{attribute addProperty BoxType "KL2809"}
{attribute addProperty Id "Channel_1Channel_E75BD82E00Channel_2Channel_E75BD82E00Channel_3Channel_E75BD82E00Channel_4Channel_E75BD82E00Channel_5Channel_E75BD82E00Channel_6Channel_E75BD82E00Channel_7Channel_E75BD82E00Channel_8Channel_E75BD82E00Channel_9Channel_E75BD82E00Channel_10Channel_E75BD82E00Channel_11Channel_E75BD82E00Channel_12Channel_E75BD82E00Channel_13Channel_E75BD82E00Channel_14Channel_E75BD82E00Channel_15Channel_E75BD82E00Channel_16Channel_E75BD82E00"}
{attribute addProperty CRC "944202743"}
{attribute addProperty SizeInBites "0"}
{attribute addProperty SizeInBytes "0"}
TYPE KL2809_384763F7 :
STRUCT
	{attribute addProperty Name "Channel_1"}
	Channel_1 : Channel_E75BD82E;
	{attribute addProperty Name "Channel_2"}
	Channel_2 : Channel_E75BD82E;
	{attribute addProperty Name "Channel_3"}
	Channel_3 : Channel_E75BD82E;
	{attribute addProperty Name "Channel_4"}
	Channel_4 : Channel_E75BD82E;
	{attribute addProperty Name "Channel_5"}
	Channel_5 : Channel_E75BD82E;
	{attribute addProperty Name "Channel_6"}
	Channel_6 : Channel_E75BD82E;
	{attribute addProperty Name "Channel_7"}
	Channel_7 : Channel_E75BD82E;
	{attribute addProperty Name "Channel_8"}
	Channel_8 : Channel_E75BD82E;
	{attribute addProperty Name "Channel_9"}
	Channel_9 : Channel_E75BD82E;
	{attribute addProperty Name "Channel_10"}
	Channel_10 : Channel_E75BD82E;
	{attribute addProperty Name "Channel_11"}
	Channel_11 : Channel_E75BD82E;
	{attribute addProperty Name "Channel_12"}
	Channel_12 : Channel_E75BD82E;
	{attribute addProperty Name "Channel_13"}
	Channel_13 : Channel_E75BD82E;
	{attribute addProperty Name "Channel_14"}
	Channel_14 : Channel_E75BD82E;
	{attribute addProperty Name "Channel_15"}
	Channel_15 : Channel_E75BD82E;
	{attribute addProperty Name "Channel_16"}
	Channel_16 : Channel_E75BD82E;
END_STRUCT
END_TYPE

(* stored: Version 1.2.0.0, ProductVersion 3.1.4024.9
   DUT KL2809_384763F7: Id {fab713f0-87d7-4d18-89ca-d41a0e1a702b} *)
